TYPE ST_VCC_NO:
STRUCT

(* A normally open valve needs permission to close! *)
(* Inputs *)
	{attribute 'pytmc' := '
	pv: CLS_SW ;
	field: ONAM CLOSE; 
	field: ZNAM OPEN;
	io: io ;
	'}
	pv_xCLS_SW	: BOOL;
	{attribute 'pytmc' := '
    pv: FORCE_CLS;
	io: io;
	'}
	pv_xOvrdCls	:	BOOL;
	{attribute 'pytmc' := '
    pv: CLS_OK;
	io: i;
	'}
	xCLS_OK	: BOOL;
	
	{attribute 'pytmc' := '
	pv: OVRD_ON;
	io: io
	'}
	xOverrideMode	:	BOOL; (* Shows the override status of this valve *)

(* Outputs *)
	{attribute 'pytmc' := '
    pv: CLS_DO;
	io: i;
	'}
	xCLS_DO	: BOOL;

END_STRUCT
END_TYPE

(* stored: Version 1.1.0.1, ProductVersion 3.1.4022.16
   DUT ST_VCC_NO: Id {b5ff0a28-38ae-4b86-b0f5-fc2738b0759d} *)
